FUNCTION_BLOCK SSC_TransferWorkpieceTo_RFC EXTENDS SSC_MoveWorkpiece_Base
VAR_INPUT
	i_ptrSSC : POINTER TO SmallSortingConveyor;
	i_ptrRFC : POINTER TO RefeedingConveyor;
END_VAR
VAR_OUTPUT
END_VAR
VAR
	m_ptrRFC : POINTER TO RefeedingConveyor;
	m_precondition:ComparisonExpression(EProcessVariables.SSC_WPAtEnd, EComparisonType.equals, EDataType.binary, TRUE, 0, '', TRUE);
	m_postcondition:ComparisonExpression(EProcessVariables.RFC_WPAtEnd, EComparisonType.equals, EDataType.binary, TRUE, 0, '', TRUE);
	m_passby : BOOL;
	m_timer : TON;
	m_switchExtended: BOOL;
	m_timerEject: TON;

END_VAR

SUPER^();

METHOD PROTECTED  AtTarget : BOOL
VAR_INPUT
END_VAR
AtTarget := FALSE;
m_ptrSSC^.METH_Switch_Extend();

IF m_ptrRFC^.WPAtStart THEN	
	m_passby := TRUE;
END_IF

IF m_passby THEN
	m_timer(IN := TRUE, PT := T#2000MS);
	IF m_timer.Q THEN
		m_ptrSSC^.METH_Switch_Retract();
		m_timer(IN := FALSE, PT := T#0MS);
		m_passby := FALSE;
		AtTarget := TRUE;
	END_IF
END_IF
END_METHOD

METHOD PROTECTED EjectOperation : BOOL
VAR_INPUT
END_VAR
EjectOperation := TRUE;
END_METHOD

METHOD FB_init : BOOL
VAR_INPUT
	bInitRetains : BOOL; // if TRUE, the retain variables are initialized (warm start / cold start)
	bInCopyCode : BOOL;  // if TRUE, the instance afterwards gets moved into the copy code (online change)
	
	i_ptrSSC: POINTER TO SmallSortingConveyor;
	i_ptrRFC: POINTER TO RefeedingConveyor;
END_VAR
m_ptrSSC := i_ptrSSC;
m_ptrRFC := i_ptrRFC;

m_id := EPrimitives.SSC_TransferWorkpieceTo_RFC;
m_timeout := T#5S;

Precondition := m_precondition;
Postcondition := m_postcondition;

FB_init := TRUE;
END_METHOD

END_FUNCTION_BLOCK

(* stored: Version 1.1.0.1
   POU SSC_TransferWorkpieceTo_RFC: Id {59e027bf-a43c-4ba6-a46a-41f7d428b2a3}, SpecialFunc None
   Method AtTarget: Id {6735a67c-01ff-4ac2-9f19-d64cedb76f61}
   Method EjectOperation: Id {c2d9b5a9-8536-4276-9381-e7be946e8c07}
   Method FB_init: Id {1cbc5fdf-41b8-4018-bb6f-4fac69d0cd22} *)
